Fanuc TP program (LS listing): MOTN022.LS

/PROG  MOTN022
/ATTR
OWNER		= MNEDITOR;
COMMENT		= "EQ EZSP2 AUF";
PROG_SIZE	= 743;
CREATE		= DATE 10-07-09  TIME 16:38:32;
MODIFIED	= DATE 16-06-13  TIME 23:05:48;
FILE_NAME	= EQPRGAPC;
VERSION		= 0;
LINE_COUNT	= 10;
MEMORY_SIZE	= 1107;
PROTECT		= READ_WRITE;
TCD:  STACK_SIZE	= 0,
      TASK_PRIORITY	= 50,
      TIME_SLICE	= 0,
      BUSY_LAMP_OFF	= 0,
      ABORT_REQUEST	= 0,
      PAUSE_REQUEST	= 0;
DEFAULT_GROUP	= 1,*,*,*,*;
CONTROL_CODE	= 00000000 00000000;
/APPL
/MN
    :  !EQ EZSP2 AUF ;
    :  !letzte  Aenderung  16.08.2011 ;
    :  R[400]=R[400]+1    ;
    :  R[819]=($SSR.$SINGLESTEP) ;
    :  $SSR.$SINGLESTEP=0 ;
    :  DO[877]=ON ;
    :  !EZ2/SP2 oeffnen ;
    :L P[1] max_speed CNT0 ACC200    ;
    :  R[819]=DO[22902]    ;
    :  $SSR.$SINGLESTEP=R[819] ;
/POS
P[1]{
   GP1:
	UF : 1, UT : 2,		CONFIG : 'N U T, 0, 0, -1',
	X =     0.000  mm,	Y =     0.000  mm,	Z =     0.000  mm,
	W =     0.000 deg,	P =     0.000 deg,	R =     0.000 deg
};
/END
